DECL E6POS XP526={X 822,Y 549,Z -255,A 0,B -90,C 180,S 6,T 16,E1 0.0,E2 0.0,E3 0.0,E4 0.0,E5 0.0,E6 0.0}
DECL FDAT FP526={TOOL_NO 4,BASE_NO 0,IPO_FRAME #BASE,POINT2[] " "}
DECL LDAT LCPDAT526={VEL 1,ACC 50.000,APO_DIST 500.000,APO_FAC 50.0000,AXIS_VEL 50.000,AXIS_ACC 50.000,ORI_TYP #VAR,CIRC_TYP #BASE,JERK_FAC 50.0000,GEAR_JERK 100.000,EXAX_IGN 0}

DECL E6POS XP527={X 772,Y 549,Z -255,A 0,B -90,C 180,S 6,T 16,E1 0.0,E2 0.0,E3 0.0,E4 0.0,E5 0.0,E6 0.0}
DECL FDAT FP527={TOOL_NO 4,BASE_NO 0,IPO_FRAME #BASE,POINT2[] " "}
DECL LDAT LCPDAT527={VEL 1,ACC 50.000,APO_DIST 500.000,APO_FAC 50.0000,AXIS_VEL 50.000,AXIS_ACC 50.000,ORI_TYP #VAR,CIRC_TYP #BASE,JERK_FAC 50.0000,GEAR_JERK 100.000,EXAX_IGN 0}

DECL E6POS XP528={X 722,Y 549,Z -255,A 0,B -90,C 180,S 6,T 16,E1 0.0,E2 0.0,E3 0.0,E4 0.0,E5 0.0,E6 0.0}
DECL FDAT FP528={TOOL_NO 4,BASE_NO 0,IPO_FRAME #BASE,POINT2[] " "}
DECL LDAT LCPDAT528={VEL 1,ACC 50.000,APO_DIST 500.000,APO_FAC 50.0000,AXIS_VEL 50.000,AXIS_ACC 50.000,ORI_TYP #VAR,CIRC_TYP #BASE,JERK_FAC 50.0000,GEAR_JERK 100.000,EXAX_IGN 0}

DECL E6POS XP529={X 672,Y 549,Z -255,A 0,B -90,C 180,S 6,T 16,E1 0.0,E2 0.0,E3 0.0,E4 0.0,E5 0.0,E6 0.0}
DECL FDAT FP529={TOOL_NO 4,BASE_NO 0,IPO_FRAME #BASE,POINT2[] " "}
DECL LDAT LCPDAT529={VEL 1,ACC 50.000,APO_DIST 500.000,APO_FAC 50.0000,AXIS_VEL 50.000,AXIS_ACC 50.000,ORI_TYP #VAR,CIRC_TYP #BASE,JERK_FAC 50.0000,GEAR_JERK 100.000,EXAX_IGN 0}

DECL E6POS XP530={X 672,Y 549,Z -205,A 0,B -90,C 180,S 6,T 16,E1 0.0,E2 0.0,E3 0.0,E4 0.0,E5 0.0,E6 0.0}
DECL FDAT FP530={TOOL_NO 4,BASE_NO 0,IPO_FRAME #BASE,POINT2[] " "}
DECL LDAT LCPDAT530={VEL 1,ACC 50.000,APO_DIST 500.000,APO_FAC 50.0000,AXIS_VEL 50.000,AXIS_ACC 50.000,ORI_TYP #VAR,CIRC_TYP #BASE,JERK_FAC 50.0000,GEAR_JERK 100.000,EXAX_IGN 0}

DECL E6POS XP531={X 722,Y 549,Z -205,A 0,B -90,C 180,S 6,T 16,E1 0.0,E2 0.0,E3 0.0,E4 0.0,E5 0.0,E6 0.0}
DECL FDAT FP531={TOOL_NO 4,BASE_NO 0,IPO_FRAME #BASE,POINT2[] " "}
DECL LDAT LCPDAT531={VEL 1,ACC 50.000,APO_DIST 500.000,APO_FAC 50.0000,AXIS_VEL 50.000,AXIS_ACC 50.000,ORI_TYP #VAR,CIRC_TYP #BASE,JERK_FAC 50.0000,GEAR_JERK 100.000,EXAX_IGN 0}

DECL E6POS XP532={X 772,Y 549,Z -205,A 0,B -90,C 180,S 6,T 16,E1 0.0,E2 0.0,E3 0.0,E4 0.0,E5 0.0,E6 0.0}
DECL FDAT FP532={TOOL_NO 4,BASE_NO 0,IPO_FRAME #BASE,POINT2[] " "}
DECL LDAT LCPDAT532={VEL 1,ACC 50.000,APO_DIST 500.000,APO_FAC 50.0000,AXIS_VEL 50.000,AXIS_ACC 50.000,ORI_TYP #VAR,CIRC_TYP #BASE,JERK_FAC 50.0000,GEAR_JERK 100.000,EXAX_IGN 0}

DECL E6POS XP533={X 822,Y 549,Z -205,A 0,B -90,C 180,S 6,T 16,E1 0.0,E2 0.0,E3 0.0,E4 0.0,E5 0.0,E6 0.0}
DECL FDAT FP533={TOOL_NO 4,BASE_NO 0,IPO_FRAME #BASE,POINT2[] " "}
DECL LDAT LCPDAT533={VEL 1,ACC 50.000,APO_DIST 500.000,APO_FAC 50.0000,AXIS_VEL 50.000,AXIS_ACC 50.000,ORI_TYP #VAR,CIRC_TYP #BASE,JERK_FAC 50.0000,GEAR_JERK 100.000,EXAX_IGN 0}

DECL E6POS XP534={X 872,Y 549,Z -205,A 0,B -90,C 180,S 6,T 16,E1 0.0,E2 0.0,E3 0.0,E4 0.0,E5 0.0,E6 0.0}
DECL FDAT FP534={TOOL_NO 4,BASE_NO 0,IPO_FRAME #BASE,POINT2[] " "}
DECL LDAT LCPDAT534={VEL 1,ACC 50.000,APO_DIST 500.000,APO_FAC 50.0000,AXIS_VEL 50.000,AXIS_ACC 50.000,ORI_TYP #VAR,CIRC_TYP #BASE,JERK_FAC 50.0000,GEAR_JERK 100.000,EXAX_IGN 0}

DECL E6POS XP535={X 922,Y 549,Z -205,A 0,B -90,C 180,S 6,T 16,E1 0.0,E2 0.0,E3 0.0,E4 0.0,E5 0.0,E6 0.0}
DECL FDAT FP535={TOOL_NO 4,BASE_NO 0,IPO_FRAME #BASE,POINT2[] " "}
DECL LDAT LCPDAT535={VEL 1,ACC 50.000,APO_DIST 500.000,APO_FAC 50.0000,AXIS_VEL 50.000,AXIS_ACC 50.000,ORI_TYP #VAR,CIRC_TYP #BASE,JERK_FAC 50.0000,GEAR_JERK 100.000,EXAX_IGN 0}

DECL E6POS XP536={X 972,Y 549,Z -205,A 0,B -90,C 180,S 6,T 16,E1 0.0,E2 0.0,E3 0.0,E4 0.0,E5 0.0,E6 0.0}
DECL FDAT FP536={TOOL_NO 4,BASE_NO 0,IPO_FRAME #BASE,POINT2[] " "}
DECL LDAT LCPDAT536={VEL 1,ACC 50.000,APO_DIST 500.000,APO_FAC 50.0000,AXIS_VEL 50.000,AXIS_ACC 50.000,ORI_TYP #VAR,CIRC_TYP #BASE,JERK_FAC 50.0000,GEAR_JERK 100.000,EXAX_IGN 0}

DECL E6POS XP537={X 1022,Y 549,Z -205,A 0,B -90,C 180,S 6,T 16,E1 0.0,E2 0.0,E3 0.0,E4 0.0,E5 0.0,E6 0.0}
DECL FDAT FP537={TOOL_NO 4,BASE_NO 0,IPO_FRAME #BASE,POINT2[] " "}
DECL LDAT LCPDAT537={VEL 1,ACC 50.000,APO_DIST 500.000,APO_FAC 50.0000,AXIS_VEL 50.000,AXIS_ACC 50.000,ORI_TYP #VAR,CIRC_TYP #BASE,JERK_FAC 50.0000,GEAR_JERK 100.000,EXAX_IGN 0}

DECL E6POS XP538={X 1072,Y 549,Z -205,A 0,B -90,C 180,S 6,T 16,E1 0.0,E2 0.0,E3 0.0,E4 0.0,E5 0.0,E6 0.0}
DECL FDAT FP538={TOOL_NO 4,BASE_NO 0,IPO_FRAME #BASE,POINT2[] " "}
DECL LDAT LCPDAT538={VEL 1,ACC 50.000,APO_DIST 500.000,APO_FAC 50.0000,AXIS_VEL 50.000,AXIS_ACC 50.000,ORI_TYP #VAR,CIRC_TYP #BASE,JERK_FAC 50.0000,GEAR_JERK 100.000,EXAX_IGN 0}

DECL E6POS XP539={X 1122,Y 549,Z -205,A 0,B -90,C 180,S 6,T 16,E1 0.0,E2 0.0,E3 0.0,E4 0.0,E5 0.0,E6 0.0}
DECL FDAT FP539={TOOL_NO 4,BASE_NO 0,IPO_FRAME #BASE,POINT2[] " "}
DECL LDAT LCPDAT539={VEL 1,ACC 50.000,APO_DIST 500.000,APO_FAC 50.0000,AXIS_VEL 50.000,AXIS_ACC 50.000,ORI_TYP #VAR,CIRC_TYP #BASE,JERK_FAC 50.0000,GEAR_JERK 100.000,EXAX_IGN 0}

DECL E6POS XP540={X 1172,Y 549,Z -205,A 0,B -90,C 180,S 6,T 16,E1 0.0,E2 0.0,E3 0.0,E4 0.0,E5 0.0,E6 0.0}
DECL FDAT FP540={TOOL_NO 4,BASE_NO 0,IPO_FRAME #BASE,POINT2[] " "}
DECL LDAT LCPDAT540={VEL 1,ACC 50.000,APO_DIST 500.000,APO_FAC 50.0000,AXIS_VEL 50.000,AXIS_ACC 50.000,ORI_TYP #VAR,CIRC_TYP #BASE,JERK_FAC 50.0000,GEAR_JERK 100.000,EXAX_IGN 0}

DECL E6POS XP541={X 1222,Y 549,Z -205,A 0,B -90,C 180,S 6,T 16,E1 0.0,E2 0.0,E3 0.0,E4 0.0,E5 0.0,E6 0.0}
DECL FDAT FP541={TOOL_NO 4,BASE_NO 0,IPO_FRAME #BASE,POINT2[] " "}
DECL LDAT LCPDAT541={VEL 1,ACC 50.000,APO_DIST 500.000,APO_FAC 50.0000,AXIS_VEL 50.000,AXIS_ACC 50.000,ORI_TYP #VAR,CIRC_TYP #BASE,JERK_FAC 50.0000,GEAR_JERK 100.000,EXAX_IGN 0}

DECL E6POS XP542={X 1272,Y 549,Z -205,A 0,B -90,C 180,S 6,T 16,E1 0.0,E2 0.0,E3 0.0,E4 0.0,E5 0.0,E6 0.0}
DECL FDAT FP542={TOOL_NO 4,BASE_NO 0,IPO_FRAME #BASE,POINT2[] " "}
DECL LDAT LCPDAT542={VEL 1,ACC 50.000,APO_DIST 500.000,APO_FAC 50.0000,AXIS_VEL 50.000,AXIS_ACC 50.000,ORI_TYP #VAR,CIRC_TYP #BASE,JERK_FAC 50.0000,GEAR_JERK 100.000,EXAX_IGN 0}

DECL E6POS XP543={X 1272,Y 549,Z -155,A 0,B -90,C 180,S 6,T 16,E1 0.0,E2 0.0,E3 0.0,E4 0.0,E5 0.0,E6 0.0}
DECL FDAT FP543={TOOL_NO 4,BASE_NO 0,IPO_FRAME #BASE,POINT2[] " "}
DECL LDAT LCPDAT543={VEL 1,ACC 50.000,APO_DIST 500.000,APO_FAC 50.0000,AXIS_VEL 50.000,AXIS_ACC 50.000,ORI_TYP #VAR,CIRC_TYP #BASE,JERK_FAC 50.0000,GEAR_JERK 100.000,EXAX_IGN 0}

DECL E6POS XP544={X 1222,Y 549,Z -155,A 0,B -90,C 180,S 6,T 16,E1 0.0,E2 0.0,E3 0.0,E4 0.0,E5 0.0,E6 0.0}
DECL FDAT FP544={TOOL_NO 4,BASE_NO 0,IPO_FRAME #BASE,POINT2[] " "}
DECL LDAT LCPDAT544={VEL 1,ACC 50.000,APO_DIST 500.000,APO_FAC 50.0000,AXIS_VEL 50.000,AXIS_ACC 50.000,ORI_TYP #VAR,CIRC_TYP #BASE,JERK_FAC 50.0000,GEAR_JERK 100.000,EXAX_IGN 0}

DECL E6POS XP545={X 1172,Y 549,Z -155,A 0,B -90,C 180,S 6,T 16,E1 0.0,E2 0.0,E3 0.0,E4 0.0,E5 0.0,E6 0.0}
DECL FDAT FP545={TOOL_NO 4,BASE_NO 0,IPO_FRAME #BASE,POINT2[] " "}
DECL LDAT LCPDAT545={VEL 1,ACC 50.000,APO_DIST 500.000,APO_FAC 50.0000,AXIS_VEL 50.000,AXIS_ACC 50.000,ORI_TYP #VAR,CIRC_TYP #BASE,JERK_FAC 50.0000,GEAR_JERK 100.000,EXAX_IGN 0}

DECL E6POS XP546={X 1122,Y 549,Z -155,A 0,B -90,C 180,S 6,T 16,E1 0.0,E2 0.0,E3 0.0,E4 0.0,E5 0.0,E6 0.0}
DECL FDAT FP546={TOOL_NO 4,BASE_NO 0,IPO_FRAME #BASE,POINT2[] " "}
DECL LDAT LCPDAT546={VEL 1,ACC 50.000,APO_DIST 500.000,APO_FAC 50.0000,AXIS_VEL 50.000,AXIS_ACC 50.000,ORI_TYP #VAR,CIRC_TYP #BASE,JERK_FAC 50.0000,GEAR_JERK 100.000,EXAX_IGN 0}

DECL E6POS XP547={X 1072,Y 549,Z -155,A 0,B -90,C 180,S 6,T 16,E1 0.0,E2 0.0,E3 0.0,E4 0.0,E5 0.0,E6 0.0}
DECL FDAT FP547={TOOL_NO 4,BASE_NO 0,IPO_FRAME #BASE,POINT2[] " "}
DECL LDAT LCPDAT547={VEL 1,ACC 50.000,APO_DIST 500.000,APO_FAC 50.0000,AXIS_VEL 50.000,AXIS_ACC 50.000,ORI_TYP #VAR,CIRC_TYP #BASE,JERK_FAC 50.0000,GEAR_JERK 100.000,EXAX_IGN 0}

DECL E6POS XP548={X 1022,Y 549,Z -155,A 0,B -90,C 180,S 6,T 16,E1 0.0,E2 0.0,E3 0.0,E4 0.0,E5 0.0,E6 0.0}
DECL FDAT FP548={TOOL_NO 4,BASE_NO 0,IPO_FRAME #BASE,POINT2[] " "}
DECL LDAT LCPDAT548={VEL 1,ACC 50.000,APO_DIST 500.000,APO_FAC 50.0000,AXIS_VEL 50.000,AXIS_ACC 50.000,ORI_TYP #VAR,CIRC_TYP #BASE,JERK_FAC 50.0000,GEAR_JERK 100.000,EXAX_IGN 0}

DECL E6POS XP549={X 972,Y 549,Z -155,A 0,B -90,C 180,S 6,T 16,E1 0.0,E2 0.0,E3 0.0,E4 0.0,E5 0.0,E6 0.0}
DECL FDAT FP549={TOOL_NO 4,BASE_NO 0,IPO_FRAME #BASE,POINT2[] " "}
DECL LDAT LCPDAT549={VEL 1,ACC 50.000,APO_DIST 500.000,APO_FAC 50.0000,AXIS_VEL 50.000,AXIS_ACC 50.000,ORI_TYP #VAR,CIRC_TYP #BASE,JERK_FAC 50.0000,GEAR_JERK 100.000,EXAX_IGN 0}

DECL E6POS XP550={X 922,Y 549,Z -155,A 0,B -90,C 180,S 6,T 16,E1 0.0,E2 0.0,E3 0.0,E4 0.0,E5 0.0,E6 0.0}
DECL FDAT FP550={TOOL_NO 4,BASE_NO 0,IPO_FRAME #BASE,POINT2[] " "}
DECL LDAT LCPDAT550={VEL 1,ACC 50.000,APO_DIST 500.000,APO_FAC 50.0000,AXIS_VEL 50.000,AXIS_ACC 50.000,ORI_TYP #VAR,CIRC_TYP #BASE,JERK_FAC 50.0000,GEAR_JERK 100.000,EXAX_IGN 0}

DECL E6POS XP551={X 872,Y 549,Z -155,A 0,B -90,C 180,S 6,T 16,E1 0.0,E2 0.0,E3 0.0,E4 0.0,E5 0.0,E6 0.0}
DECL FDAT FP551={TOOL_NO 4,BASE_NO 0,IPO_FRAME #BASE,POINT2[] " "}
DECL LDAT LCPDAT551={VEL 1,ACC 50.000,APO_DIST 500.000,APO_FAC 50.0000,AXIS_VEL 50.000,AXIS_ACC 50.000,ORI_TYP #VAR,CIRC_TYP #BASE,JERK_FAC 50.0000,GEAR_JERK 100.000,EXAX_IGN 0}

DECL E6POS XP552={X 822,Y 549,Z -155,A 0,B -90,C 180,S 6,T 16,E1 0.0,E2 0.0,E3 0.0,E4 0.0,E5 0.0,E6 0.0}
DECL FDAT FP552={TOOL_NO 4,BASE_NO 0,IPO_FRAME #BASE,POINT2[] " "}
DECL LDAT LCPDAT552={VEL 1,ACC 50.000,APO_DIST 500.000,APO_FAC 50.0000,AXIS_VEL 50.000,AXIS_ACC 50.000,ORI_TYP #VAR,CIRC_TYP #BASE,JERK_FAC 50.0000,GEAR_JERK 100.000,EXAX_IGN 0}

DECL E6POS XP553={X 772,Y 549,Z -155,A 0,B -90,C 180,S 6,T 16,E1 0.0,E2 0.0,E3 0.0,E4 0.0,E5 0.0,E6 0.0}
DECL FDAT FP553={TOOL_NO 4,BASE_NO 0,IPO_FRAME #BASE,POINT2[] " "}
DECL LDAT LCPDAT553={VEL 1,ACC 50.000,APO_DIST 500.000,APO_FAC 50.0000,AXIS_VEL 50.000,AXIS_ACC 50.000,ORI_TYP #VAR,CIRC_TYP #BASE,JERK_FAC 50.0000,GEAR_JERK 100.000,EXAX_IGN 0}

DECL E6POS XP554={X 722,Y 549,Z -155,A 0,B -90,C 180,S 6,T 16,E1 0.0,E2 0.0,E3 0.0,E4 0.0,E5 0.0,E6 0.0}
DECL FDAT FP554={TOOL_NO 4,BASE_NO 0,IPO_FRAME #BASE,POINT2[] " "}
DECL LDAT LCPDAT554={VEL 1,ACC 50.000,APO_DIST 500.000,APO_FAC 50.0000,AXIS_VEL 50.000,AXIS_ACC 50.000,ORI_TYP #VAR,CIRC_TYP #BASE,JERK_FAC 50.0000,GEAR_JERK 100.000,EXAX_IGN 0}

DECL E6POS XP555={X 672,Y 549,Z -155,A 0,B -90,C 180,S 6,T 16,E1 0.0,E2 0.0,E3 0.0,E4 0.0,E5 0.0,E6 0.0}
DECL FDAT FP555={TOOL_NO 4,BASE_NO 0,IPO_FRAME #BASE,POINT2[] " "}
DECL LDAT LCPDAT555={VEL 1,ACC 50.000,APO_DIST 500.000,APO_FAC 50.0000,AXIS_VEL 50.000,AXIS_ACC 50.000,ORI_TYP #VAR,CIRC_TYP #BASE,JERK_FAC 50.0000,GEAR_JERK 100.000,EXAX_IGN 0}

DECL E6POS XP556={X 672,Y 549,Z -105,A 0,B -90,C 180,S 6,T 16,E1 0.0,E2 0.0,E3 0.0,E4 0.0,E5 0.0,E6 0.0}
DECL FDAT FP556={TOOL_NO 4,BASE_NO 0,IPO_FRAME #BASE,POINT2[] " "}
DECL LDAT LCPDAT556={VEL 1,ACC 50.000,APO_DIST 500.000,APO_FAC 50.0000,AXIS_VEL 50.000,AXIS_ACC 50.000,ORI_TYP #VAR,CIRC_TYP #BASE,JERK_FAC 50.0000,GEAR_JERK 100.000,EXAX_IGN 0}

DECL E6POS XP557={X 722,Y 549,Z -105,A 0,B -90,C 180,S 6,T 16,E1 0.0,E2 0.0,E3 0.0,E4 0.0,E5 0.0,E6 0.0}
DECL FDAT FP557={TOOL_NO 4,BASE_NO 0,IPO_FRAME #BASE,POINT2[] " "}
DECL LDAT LCPDAT557={VEL 1,ACC 50.000,APO_DIST 500.000,APO_FAC 50.0000,AXIS_VEL 50.000,AXIS_ACC 50.000,ORI_TYP #VAR,CIRC_TYP #BASE,JERK_FAC 50.0000,GEAR_JERK 100.000,EXAX_IGN 0}

DECL E6POS XP558={X 772,Y 549,Z -105,A 0,B -90,C 180,S 6,T 16,E1 0.0,E2 0.0,E3 0.0,E4 0.0,E5 0.0,E6 0.0}
DECL FDAT FP558={TOOL_NO 4,BASE_NO 0,IPO_FRAME #BASE,POINT2[] " "}
DECL LDAT LCPDAT558={VEL 1,ACC 50.000,APO_DIST 500.000,APO_FAC 50.0000,AXIS_VEL 50.000,AXIS_ACC 50.000,ORI_TYP #VAR,CIRC_TYP #BASE,JERK_FAC 50.0000,GEAR_JERK 100.000,EXAX_IGN 0}

DECL E6POS XP559={X 822,Y 549,Z -105,A 0,B -90,C 180,S 6,T 16,E1 0.0,E2 0.0,E3 0.0,E4 0.0,E5 0.0,E6 0.0}
DECL FDAT FP559={TOOL_NO 4,BASE_NO 0,IPO_FRAME #BASE,POINT2[] " "}
DECL LDAT LCPDAT559={VEL 1,ACC 50.000,APO_DIST 500.000,APO_FAC 50.0000,AXIS_VEL 50.000,AXIS_ACC 50.000,ORI_TYP #VAR,CIRC_TYP #BASE,JERK_FAC 50.0000,GEAR_JERK 100.000,EXAX_IGN 0}

DECL E6POS XP560={X 872,Y 549,Z -105,A 0,B -90,C 180,S 6,T 16,E1 0.0,E2 0.0,E3 0.0,E4 0.0,E5 0.0,E6 0.0}
DECL FDAT FP560={TOOL_NO 4,BASE_NO 0,IPO_FRAME #BASE,POINT2[] " "}
DECL LDAT LCPDAT560={VEL 1,ACC 50.000,APO_DIST 500.000,APO_FAC 50.0000,AXIS_VEL 50.000,AXIS_ACC 50.000,ORI_TYP #VAR,CIRC_TYP #BASE,JERK_FAC 50.0000,GEAR_JERK 100.000,EXAX_IGN 0}

DECL E6POS XP561={X 922,Y 549,Z -105,A 0,B -90,C 180,S 6,T 16,E1 0.0,E2 0.0,E3 0.0,E4 0.0,E5 0.0,E6 0.0}
DECL FDAT FP561={TOOL_NO 4,BASE_NO 0,IPO_FRAME #BASE,POINT2[] " "}
DECL LDAT LCPDAT561={VEL 1,ACC 50.000,APO_DIST 500.000,APO_FAC 50.0000,AXIS_VEL 50.000,AXIS_ACC 50.000,ORI_TYP #VAR,CIRC_TYP #BASE,JERK_FAC 50.0000,GEAR_JERK 100.000,EXAX_IGN 0}

DECL E6POS XP562={X 972,Y 549,Z -105,A 0,B -90,C 180,S 6,T 16,E1 0.0,E2 0.0,E3 0.0,E4 0.0,E5 0.0,E6 0.0}
DECL FDAT FP562={TOOL_NO 4,BASE_NO 0,IPO_FRAME #BASE,POINT2[] " "}
DECL LDAT LCPDAT562={VEL 1,ACC 50.000,APO_DIST 500.000,APO_FAC 50.0000,AXIS_VEL 50.000,AXIS_ACC 50.000,ORI_TYP #VAR,CIRC_TYP #BASE,JERK_FAC 50.0000,GEAR_JERK 100.000,EXAX_IGN 0}

DECL E6POS XP563={X 1022,Y 549,Z -105,A 0,B -90,C 180,S 6,T 16,E1 0.0,E2 0.0,E3 0.0,E4 0.0,E5 0.0,E6 0.0}
DECL FDAT FP563={TOOL_NO 4,BASE_NO 0,IPO_FRAME #BASE,POINT2[] " "}
DECL LDAT LCPDAT563={VEL 1,ACC 50.000,APO_DIST 500.000,APO_FAC 50.0000,AXIS_VEL 50.000,AXIS_ACC 50.000,ORI_TYP #VAR,CIRC_TYP #BASE,JERK_FAC 50.0000,GEAR_JERK 100.000,EXAX_IGN 0}

DECL E6POS XP564={X 1072,Y 549,Z -105,A 0,B -90,C 180,S 6,T 16,E1 0.0,E2 0.0,E3 0.0,E4 0.0,E5 0.0,E6 0.0}
DECL FDAT FP564={TOOL_NO 4,BASE_NO 0,IPO_FRAME #BASE,POINT2[] " "}
DECL LDAT LCPDAT564={VEL 1,ACC 50.000,APO_DIST 500.000,APO_FAC 50.0000,AXIS_VEL 50.000,AXIS_ACC 50.000,ORI_TYP #VAR,CIRC_TYP #BASE,JERK_FAC 50.0000,GEAR_JERK 100.000,EXAX_IGN 0}

DECL E6POS XP565={X 1122,Y 549,Z -105,A 0,B -90,C 180,S 6,T 16,E1 0.0,E2 0.0,E3 0.0,E4 0.0,E5 0.0,E6 0.0}
DECL FDAT FP565={TOOL_NO 4,BASE_NO 0,IPO_FRAME #BASE,POINT2[] " "}
DECL LDAT LCPDAT565={VEL 1,ACC 50.000,APO_DIST 500.000,APO_FAC 50.0000,AXIS_VEL 50.000,AXIS_ACC 50.000,ORI_TYP #VAR,CIRC_TYP #BASE,JERK_FAC 50.0000,GEAR_JERK 100.000,EXAX_IGN 0}

DECL E6POS XP566={X 1172,Y 549,Z -105,A 0,B -90,C 180,S 6,T 16,E1 0.0,E2 0.0,E3 0.0,E4 0.0,E5 0.0,E6 0.0}
DECL FDAT FP566={TOOL_NO 4,BASE_NO 0,IPO_FRAME #BASE,POINT2[] " "}
DECL LDAT LCPDAT566={VEL 1,ACC 50.000,APO_DIST 500.000,APO_FAC 50.0000,AXIS_VEL 50.000,AXIS_ACC 50.000,ORI_TYP #VAR,CIRC_TYP #BASE,JERK_FAC 50.0000,GEAR_JERK 100.000,EXAX_IGN 0}

DECL E6POS XP567={X 1222,Y 549,Z -105,A 0,B -90,C 180,S 6,T 16,E1 0.0,E2 0.0,E3 0.0,E4 0.0,E5 0.0,E6 0.0}
DECL FDAT FP567={TOOL_NO 4,BASE_NO 0,IPO_FRAME #BASE,POINT2[] " "}
DECL LDAT LCPDAT567={VEL 1,ACC 50.000,APO_DIST 500.000,APO_FAC 50.0000,AXIS_VEL 50.000,AXIS_ACC 50.000,ORI_TYP #VAR,CIRC_TYP #BASE,JERK_FAC 50.0000,GEAR_JERK 100.000,EXAX_IGN 0}

DECL E6POS XP568={X 1272,Y 549,Z -105,A 0,B -90,C 180,S 6,T 16,E1 0.0,E2 0.0,E3 0.0,E4 0.0,E5 0.0,E6 0.0}
DECL FDAT FP568={TOOL_NO 4,BASE_NO 0,IPO_FRAME #BASE,POINT2[] " "}
DECL LDAT LCPDAT568={VEL 1,ACC 50.000,APO_DIST 500.000,APO_FAC 50.0000,AXIS_VEL 50.000,AXIS_ACC 50.000,ORI_TYP #VAR,CIRC_TYP #BASE,JERK_FAC 50.0000,GEAR_JERK 100.000,EXAX_IGN 0}

DECL E6POS XP569={X 1272,Y 549,Z -55,A 0,B -90,C 180,S 6,T 16,E1 0.0,E2 0.0,E3 0.0,E4 0.0,E5 0.0,E6 0.0}
DECL FDAT FP569={TOOL_NO 4,BASE_NO 0,IPO_FRAME #BASE,POINT2[] " "}
DECL LDAT LCPDAT569={VEL 1,ACC 50.000,APO_DIST 500.000,APO_FAC 50.0000,AXIS_VEL 50.000,AXIS_ACC 50.000,ORI_TYP #VAR,CIRC_TYP #BASE,JERK_FAC 50.0000,GEAR_JERK 100.000,EXAX_IGN 0}

DECL E6POS XP570={X 1222,Y 549,Z -55,A 0,B -90,C 180,S 6,T 16,E1 0.0,E2 0.0,E3 0.0,E4 0.0,E5 0.0,E6 0.0}
DECL FDAT FP570={TOOL_NO 4,BASE_NO 0,IPO_FRAME #BASE,POINT2[] " "}
DECL LDAT LCPDAT570={VEL 1,ACC 50.000,APO_DIST 500.000,APO_FAC 50.0000,AXIS_VEL 50.000,AXIS_ACC 50.000,ORI_TYP #VAR,CIRC_TYP #BASE,JERK_FAC 50.0000,GEAR_JERK 100.000,EXAX_IGN 0}

DECL E6POS XP571={X 1172,Y 549,Z -55,A 0,B -90,C 180,S 6,T 16,E1 0.0,E2 0.0,E3 0.0,E4 0.0,E5 0.0,E6 0.0}
DECL FDAT FP571={TOOL_NO 4,BASE_NO 0,IPO_FRAME #BASE,POINT2[] " "}
DECL LDAT LCPDAT571={VEL 1,ACC 50.000,APO_DIST 500.000,APO_FAC 50.0000,AXIS_VEL 50.000,AXIS_ACC 50.000,ORI_TYP #VAR,CIRC_TYP #BASE,JERK_FAC 50.0000,GEAR_JERK 100.000,EXAX_IGN 0}

DECL E6POS XP572={X 1122,Y 549,Z -55,A 0,B -90,C 180,S 6,T 16,E1 0.0,E2 0.0,E3 0.0,E4 0.0,E5 0.0,E6 0.0}
DECL FDAT FP572={TOOL_NO 4,BASE_NO 0,IPO_FRAME #BASE,POINT2[] " "}
DECL LDAT LCPDAT572={VEL 1,ACC 50.000,APO_DIST 500.000,APO_FAC 50.0000,AXIS_VEL 50.000,AXIS_ACC 50.000,ORI_TYP #VAR,CIRC_TYP #BASE,JERK_FAC 50.0000,GEAR_JERK 100.000,EXAX_IGN 0}

DECL E6POS XP573={X 1072,Y 549,Z -55,A 0,B -90,C 180,S 6,T 16,E1 0.0,E2 0.0,E3 0.0,E4 0.0,E5 0.0,E6 0.0}
DECL FDAT FP573={TOOL_NO 4,BASE_NO 0,IPO_FRAME #BASE,POINT2[] " "}
DECL LDAT LCPDAT573={VEL 1,ACC 50.000,APO_DIST 500.000,APO_FAC 50.0000,AXIS_VEL 50.000,AXIS_ACC 50.000,ORI_TYP #VAR,CIRC_TYP #BASE,JERK_FAC 50.0000,GEAR_JERK 100.000,EXAX_IGN 0}

DECL E6POS XP574={X 1022,Y 549,Z -55,A 0,B -90,C 180,S 6,T 16,E1 0.0,E2 0.0,E3 0.0,E4 0.0,E5 0.0,E6 0.0}
DECL FDAT FP574={TOOL_NO 4,BASE_NO 0,IPO_FRAME #BASE,POINT2[] " "}
DECL LDAT LCPDAT574={VEL 1,ACC 50.000,APO_DIST 500.000,APO_FAC 50.0000,AXIS_VEL 50.000,AXIS_ACC 50.000,ORI_TYP #VAR,CIRC_TYP #BASE,JERK_FAC 50.0000,GEAR_JERK 100.000,EXAX_IGN 0}

DECL E6POS XP575={X 972,Y 549,Z -55,A 0,B -90,C 180,S 6,T 16,E1 0.0,E2 0.0,E3 0.0,E4 0.0,E5 0.0,E6 0.0}
DECL FDAT FP575={TOOL_NO 4,BASE_NO 0,IPO_FRAME #BASE,POINT2[] " "}
DECL LDAT LCPDAT575={VEL 1,ACC 50.000,APO_DIST 500.000,APO_FAC 50.0000,AXIS_VEL 50.000,AXIS_ACC 50.000,ORI_TYP #VAR,CIRC_TYP #BASE,JERK_FAC 50.0000,GEAR_JERK 100.000,EXAX_IGN 0}

DECL E6POS XP576={X 922,Y 549,Z -55,A 0,B -90,C 180,S 6,T 16,E1 0.0,E2 0.0,E3 0.0,E4 0.0,E5 0.0,E6 0.0}
DECL FDAT FP576={TOOL_NO 4,BASE_NO 0,IPO_FRAME #BASE,POINT2[] " "}
DECL LDAT LCPDAT576={VEL 1,ACC 50.000,APO_DIST 500.000,APO_FAC 50.0000,AXIS_VEL 50.000,AXIS_ACC 50.000,ORI_TYP #VAR,CIRC_TYP #BASE,JERK_FAC 50.0000,GEAR_JERK 100.000,EXAX_IGN 0}

DECL E6POS XP577={X 872,Y 549,Z -55,A 0,B -90,C 180,S 6,T 16,E1 0.0,E2 0.0,E3 0.0,E4 0.0,E5 0.0,E6 0.0}
DECL FDAT FP577={TOOL_NO 4,BASE_NO 0,IPO_FRAME #BASE,POINT2[] " "}
DECL LDAT LCPDAT577={VEL 1,ACC 50.000,APO_DIST 500.000,APO_FAC 50.0000,AXIS_VEL 50.000,AXIS_ACC 50.000,ORI_TYP #VAR,CIRC_TYP #BASE,JERK_FAC 50.0000,GEAR_JERK 100.000,EXAX_IGN 0}

DECL E6POS XP578={X 822,Y 549,Z -55,A 0,B -90,C 180,S 6,T 16,E1 0.0,E2 0.0,E3 0.0,E4 0.0,E5 0.0,E6 0.0}
DECL FDAT FP578={TOOL_NO 4,BASE_NO 0,IPO_FRAME #BASE,POINT2[] " "}
DECL LDAT LCPDAT578={VEL 1,ACC 50.000,APO_DIST 500.000,APO_FAC 50.0000,AXIS_VEL 50.000,AXIS_ACC 50.000,ORI_TYP #VAR,CIRC_TYP #BASE,JERK_FAC 50.0000,GEAR_JERK 100.000,EXAX_IGN 0}

DECL E6POS XP579={X 772,Y 549,Z -55,A 0,B -90,C 180,S 6,T 16,E1 0.0,E2 0.0,E3 0.0,E4 0.0,E5 0.0,E6 0.0}
DECL FDAT FP579={TOOL_NO 4,BASE_NO 0,IPO_FRAME #BASE,POINT2[] " "}
DECL LDAT LCPDAT579={VEL 1,ACC 50.000,APO_DIST 500.000,APO_FAC 50.0000,AXIS_VEL 50.000,AXIS_ACC 50.000,ORI_TYP #VAR,CIRC_TYP #BASE,JERK_FAC 50.0000,GEAR_JERK 100.000,EXAX_IGN 0}

DECL E6POS XP580={X 722,Y 549,Z -55,A 0,B -90,C 180,S 6,T 16,E1 0.0,E2 0.0,E3 0.0,E4 0.0,E5 0.0,E6 0.0}
DECL FDAT FP580={TOOL_NO 4,BASE_NO 0,IPO_FRAME #BASE,POINT2[] " "}
DECL LDAT LCPDAT580={VEL 1,ACC 50.000,APO_DIST 500.000,APO_FAC 50.0000,AXIS_VEL 50.000,AXIS_ACC 50.000,ORI_TYP #VAR,CIRC_TYP #BASE,JERK_FAC 50.0000,GEAR_JERK 100.000,EXAX_IGN 0}

DECL E6POS XP581={X 672,Y 549,Z -55,A 0,B -90,C 180,S 6,T 16,E1 0.0,E2 0.0,E3 0.0,E4 0.0,E5 0.0,E6 0.0}
DECL FDAT FP581={TOOL_NO 4,BASE_NO 0,IPO_FRAME #BASE,POINT2[] " "}
DECL LDAT LCPDAT581={VEL 1,ACC 50.000,APO_DIST 500.000,APO_FAC 50.0000,AXIS_VEL 50.000,AXIS_ACC 50.000,ORI_TYP #VAR,CIRC_TYP #BASE,JERK_FAC 50.0000,GEAR_JERK 100.000,EXAX_IGN 0}

DECL E6POS XP582={X 672,Y 549,Z -5,A 0,B -90,C 180,S 6,T 16,E1 0.0,E2 0.0,E3 0.0,E4 0.0,E5 0.0,E6 0.0}
DECL FDAT FP582={TOOL_NO 4,BASE_NO 0,IPO_FRAME #BASE,POINT2[] " "}
DECL LDAT LCPDAT582={VEL 1,ACC 50.000,APO_DIST 500.000,APO_FAC 50.0000,AXIS_VEL 50.000,AXIS_ACC 50.000,ORI_TYP #VAR,CIRC_TYP #BASE,JERK_FAC 50.0000,GEAR_JERK 100.000,EXAX_IGN 0}

DECL E6POS XP583={X 722,Y 549,Z -5,A 0,B -90,C 180,S 6,T 16,E1 0.0,E2 0.0,E3 0.0,E4 0.0,E5 0.0,E6 0.0}
DECL FDAT FP583={TOOL_NO 4,BASE_NO 0,IPO_FRAME #BASE,POINT2[] " "}
DECL LDAT LCPDAT583={VEL 1,ACC 50.000,APO_DIST 500.000,APO_FAC 50.0000,AXIS_VEL 50.000,AXIS_ACC 50.000,ORI_TYP #VAR,CIRC_TYP #BASE,JERK_FAC 50.0000,GEAR_JERK 100.000,EXAX_IGN 0}

DECL E6POS XP584={X 772,Y 549,Z -5,A 0,B -90,C 180,S 6,T 16,E1 0.0,E2 0.0,E3 0.0,E4 0.0,E5 0.0,E6 0.0}
DECL FDAT FP584={TOOL_NO 4,BASE_NO 0,IPO_FRAME #BASE,POINT2[] " "}
DECL LDAT LCPDAT584={VEL 1,ACC 50.000,APO_DIST 500.000,APO_FAC 50.0000,AXIS_VEL 50.000,AXIS_ACC 50.000,ORI_TYP #VAR,CIRC_TYP #BASE,JERK_FAC 50.0000,GEAR_JERK 100.000,EXAX_IGN 0}

DECL E6POS XP585={X 822,Y 549,Z -5,A 0,B -90,C 180,S 6,T 16,E1 0.0,E2 0.0,E3 0.0,E4 0.0,E5 0.0,E6 0.0}
DECL FDAT FP585={TOOL_NO 4,BASE_NO 0,IPO_FRAME #BASE,POINT2[] " "}
DECL LDAT LCPDAT585={VEL 1,ACC 50.000,APO_DIST 500.000,APO_FAC 50.0000,AXIS_VEL 50.000,AXIS_ACC 50.000,ORI_TYP #VAR,CIRC_TYP #BASE,JERK_FAC 50.0000,GEAR_JERK 100.000,EXAX_IGN 0}

DECL E6POS XP586={X 872,Y 549,Z -5,A 0,B -90,C 180,S 6,T 16,E1 0.0,E2 0.0,E3 0.0,E4 0.0,E5 0.0,E6 0.0}
DECL FDAT FP586={TOOL_NO 4,BASE_NO 0,IPO_FRAME #BASE,POINT2[] " "}
DECL LDAT LCPDAT586={VEL 1,ACC 50.000,APO_DIST 500.000,APO_FAC 50.0000,AXIS_VEL 50.000,AXIS_ACC 50.000,ORI_TYP #VAR,CIRC_TYP #BASE,JERK_FAC 50.0000,GEAR_JERK 100.000,EXAX_IGN 0}

DECL E6POS XP587={X 922,Y 549,Z -5,A 0,B -90,C 180,S 6,T 16,E1 0.0,E2 0.0,E3 0.0,E4 0.0,E5 0.0,E6 0.0}
DECL FDAT FP587={TOOL_NO 4,BASE_NO 0,IPO_FRAME #BASE,POINT2[] " "}
DECL LDAT LCPDAT587={VEL 1,ACC 50.000,APO_DIST 500.000,APO_FAC 50.0000,AXIS_VEL 50.000,AXIS_ACC 50.000,ORI_TYP #VAR,CIRC_TYP #BASE,JERK_FAC 50.0000,GEAR_JERK 100.000,EXAX_IGN 0}

DECL E6POS XP588={X 972,Y 549,Z -5,A 0,B -90,C 180,S 6,T 16,E1 0.0,E2 0.0,E3 0.0,E4 0.0,E5 0.0,E6 0.0}
DECL FDAT FP588={TOOL_NO 4,BASE_NO 0,IPO_FRAME #BASE,POINT2[] " "}
DECL LDAT LCPDAT588={VEL 1,ACC 50.000,APO_DIST 500.000,APO_FAC 50.0000,AXIS_VEL 50.000,AXIS_ACC 50.000,ORI_TYP #VAR,CIRC_TYP #BASE,JERK_FAC 50.0000,GEAR_JERK 100.000,EXAX_IGN 0}

DECL E6POS XP589={X 1022,Y 549,Z -5,A 0,B -90,C 180,S 6,T 16,E1 0.0,E2 0.0,E3 0.0,E4 0.0,E5 0.0,E6 0.0}
DECL FDAT FP589={TOOL_NO 4,BASE_NO 0,IPO_FRAME #BASE,POINT2[] " "}
DECL LDAT LCPDAT589={VEL 1,ACC 50.000,APO_DIST 500.000,APO_FAC 50.0000,AXIS_VEL 50.000,AXIS_ACC 50.000,ORI_TYP #VAR,CIRC_TYP #BASE,JERK_FAC 50.0000,GEAR_JERK 100.000,EXAX_IGN 0}

DECL E6POS XP590={X 1072,Y 549,Z -5,A 0,B -90,C 180,S 6,T 16,E1 0.0,E2 0.0,E3 0.0,E4 0.0,E5 0.0,E6 0.0}
DECL FDAT FP590={TOOL_NO 4,BASE_NO 0,IPO_FRAME #BASE,POINT2[] " "}
DECL LDAT LCPDAT590={VEL 1,ACC 50.000,APO_DIST 500.000,APO_FAC 50.0000,AXIS_VEL 50.000,AXIS_ACC 50.000,ORI_TYP #VAR,CIRC_TYP #BASE,JERK_FAC 50.0000,GEAR_JERK 100.000,EXAX_IGN 0}

DECL E6POS XP591={X 1122,Y 549,Z -5,A 0,B -90,C 180,S 6,T 16,E1 0.0,E2 0.0,E3 0.0,E4 0.0,E5 0.0,E6 0.0}
DECL FDAT FP591={TOOL_NO 4,BASE_NO 0,IPO_FRAME #BASE,POINT2[] " "}
DECL LDAT LCPDAT591={VEL 1,ACC 50.000,APO_DIST 500.000,APO_FAC 50.0000,AXIS_VEL 50.000,AXIS_ACC 50.000,ORI_TYP #VAR,CIRC_TYP #BASE,JERK_FAC 50.0000,GEAR_JERK 100.000,EXAX_IGN 0}

DECL E6POS XP592={X 1172,Y 549,Z -5,A 0,B -90,C 180,S 6,T 16,E1 0.0,E2 0.0,E3 0.0,E4 0.0,E5 0.0,E6 0.0}
DECL FDAT FP592={TOOL_NO 4,BASE_NO 0,IPO_FRAME #BASE,POINT2[] " "}
DECL LDAT LCPDAT592={VEL 1,ACC 50.000,APO_DIST 500.000,APO_FAC 50.0000,AXIS_VEL 50.000,AXIS_ACC 50.000,ORI_TYP #VAR,CIRC_TYP #BASE,JERK_FAC 50.0000,GEAR_JERK 100.000,EXAX_IGN 0}

DECL E6POS XP593={X 1222,Y 549,Z -5,A 0,B -90,C 180,S 6,T 16,E1 0.0,E2 0.0,E3 0.0,E4 0.0,E5 0.0,E6 0.0}
DECL FDAT FP593={TOOL_NO 4,BASE_NO 0,IPO_FRAME #BASE,POINT2[] " "}
DECL LDAT LCPDAT593={VEL 1,ACC 50.000,APO_DIST 500.000,APO_FAC 50.0000,AXIS_VEL 50.000,AXIS_ACC 50.000,ORI_TYP #VAR,CIRC_TYP #BASE,JERK_FAC 50.0000,GEAR_JERK 100.000,EXAX_IGN 0}

DECL E6POS XP594={X 1272,Y 549,Z -5,A 0,B -90,C 180,S 6,T 16,E1 0.0,E2 0.0,E3 0.0,E4 0.0,E5 0.0,E6 0.0}
DECL FDAT FP594={TOOL_NO 4,BASE_NO 0,IPO_FRAME #BASE,POINT2[] " "}
DECL LDAT LCPDAT594={VEL 1,ACC 50.000,APO_DIST 500.000,APO_FAC 50.0000,AXIS_VEL 50.000,AXIS_ACC 50.000,ORI_TYP #VAR,CIRC_TYP #BASE,JERK_FAC 50.0000,GEAR_JERK 100.000,EXAX_IGN 0}

DECL E6POS XP595={X 1272,Y 549,Z 45,A 0,B -90,C 180,S 6,T 16,E1 0.0,E2 0.0,E3 0.0,E4 0.0,E5 0.0,E6 0.0}
DECL FDAT FP595={TOOL_NO 4,BASE_NO 0,IPO_FRAME #BASE,POINT2[] " "}
DECL LDAT LCPDAT595={VEL 1,ACC 50.000,APO_DIST 500.000,APO_FAC 50.0000,AXIS_VEL 50.000,AXIS_ACC 50.000,ORI_TYP #VAR,CIRC_TYP #BASE,JERK_FAC 50.0000,GEAR_JERK 100.000,EXAX_IGN 0}

DECL E6POS XP596={X 1222,Y 549,Z 45,A 0,B -90,C 180,S 6,T 16,E1 0.0,E2 0.0,E3 0.0,E4 0.0,E5 0.0,E6 0.0}
DECL FDAT FP596={TOOL_NO 4,BASE_NO 0,IPO_FRAME #BASE,POINT2[] " "}
DECL LDAT LCPDAT596={VEL 1,ACC 50.000,APO_DIST 500.000,APO_FAC 50.0000,AXIS_VEL 50.000,AXIS_ACC 50.000,ORI_TYP #VAR,CIRC_TYP #BASE,JERK_FAC 50.0000,GEAR_JERK 100.000,EXAX_IGN 0}

DECL E6POS XP597={X 1172,Y 549,Z 45,A 0,B -90,C 180,S 6,T 16,E1 0.0,E2 0.0,E3 0.0,E4 0.0,E5 0.0,E6 0.0}
DECL FDAT FP597={TOOL_NO 4,BASE_NO 0,IPO_FRAME #BASE,POINT2[] " "}
DECL LDAT LCPDAT597={VEL 1,ACC 50.000,APO_DIST 500.000,APO_FAC 50.0000,AXIS_VEL 50.000,AXIS_ACC 50.000,ORI_TYP #VAR,CIRC_TYP #BASE,JERK_FAC 50.0000,GEAR_JERK 100.000,EXAX_IGN 0}

DECL E6POS XP598={X 1122,Y 549,Z 45,A 0,B -90,C 180,S 6,T 16,E1 0.0,E2 0.0,E3 0.0,E4 0.0,E5 0.0,E6 0.0}
DECL FDAT FP598={TOOL_NO 4,BASE_NO 0,IPO_FRAME #BASE,POINT2[] " "}
DECL LDAT LCPDAT598={VEL 1,ACC 50.000,APO_DIST 500.000,APO_FAC 50.0000,AXIS_VEL 50.000,AXIS_ACC 50.000,ORI_TYP #VAR,CIRC_TYP #BASE,JERK_FAC 50.0000,GEAR_JERK 100.000,EXAX_IGN 0}

DECL E6POS XP599={X 1072,Y 549,Z 45,A 0,B -90,C 180,S 6,T 16,E1 0.0,E2 0.0,E3 0.0,E4 0.0,E5 0.0,E6 0.0}
DECL FDAT FP599={TOOL_NO 4,BASE_NO 0,IPO_FRAME #BASE,POINT2[] " "}
DECL LDAT LCPDAT599={VEL 1,ACC 50.000,APO_DIST 500.000,APO_FAC 50.0000,AXIS_VEL 50.000,AXIS_ACC 50.000,ORI_TYP #VAR,CIRC_TYP #BASE,JERK_FAC 50.0000,GEAR_JERK 100.000,EXAX_IGN 0}

DECL E6POS XP600={X 1022,Y 549,Z 45,A 0,B -90,C 180,S 6,T 16,E1 0.0,E2 0.0,E3 0.0,E4 0.0,E5 0.0,E6 0.0}
DECL FDAT FP600={TOOL_NO 4,BASE_NO 0,IPO_FRAME #BASE,POINT2[] " "}
DECL LDAT LCPDAT600={VEL 1,ACC 50.000,APO_DIST 500.000,APO_FAC 50.0000,AXIS_VEL 50.000,AXIS_ACC 50.000,ORI_TYP #VAR,CIRC_TYP #BASE,JERK_FAC 50.0000,GEAR_JERK 100.000,EXAX_IGN 0}

DECL E6POS XP601={X 972,Y 549,Z 45,A 0,B -90,C 180,S 6,T 16,E1 0.0,E2 0.0,E3 0.0,E4 0.0,E5 0.0,E6 0.0}
DECL FDAT FP601={TOOL_NO 4,BASE_NO 0,IPO_FRAME #BASE,POINT2[] " "}
DECL LDAT LCPDAT601={VEL 1,ACC 50.000,APO_DIST 500.000,APO_FAC 50.0000,AXIS_VEL 50.000,AXIS_ACC 50.000,ORI_TYP #VAR,CIRC_TYP #BASE,JERK_FAC 50.0000,GEAR_JERK 100.000,EXAX_IGN 0}

DECL E6POS XP602={X 922,Y 549,Z 45,A 0,B -90,C 180,S 6,T 16,E1 0.0,E2 0.0,E3 0.0,E4 0.0,E5 0.0,E6 0.0}
DECL FDAT FP602={TOOL_NO 4,BASE_NO 0,IPO_FRAME #BASE,POINT2[] " "}
DECL LDAT LCPDAT602={VEL 1,ACC 50.000,APO_DIST 500.000,APO_FAC 50.0000,AXIS_VEL 50.000,AXIS_ACC 50.000,ORI_TYP #VAR,CIRC_TYP #BASE,JERK_FAC 50.0000,GEAR_JERK 100.000,EXAX_IGN 0}

DECL E6POS XP603={X 872,Y 549,Z 45,A 0,B -90,C 180,S 6,T 16,E1 0.0,E2 0.0,E3 0.0,E4 0.0,E5 0.0,E6 0.0}
DECL FDAT FP603={TOOL_NO 4,BASE_NO 0,IPO_FRAME #BASE,POINT2[] " "}
DECL LDAT LCPDAT603={VEL 1,ACC 50.000,APO_DIST 500.000,APO_FAC 50.0000,AXIS_VEL 50.000,AXIS_ACC 50.000,ORI_TYP #VAR,CIRC_TYP #BASE,JERK_FAC 50.0000,GEAR_JERK 100.000,EXAX_IGN 0}

DECL E6POS XP604={X 822,Y 549,Z 45,A 0,B -90,C 180,S 6,T 16,E1 0.0,E2 0.0,E3 0.0,E4 0.0,E5 0.0,E6 0.0}
DECL FDAT FP604={TOOL_NO 4,BASE_NO 0,IPO_FRAME #BASE,POINT2[] " "}
DECL LDAT LCPDAT604={VEL 1,ACC 50.000,APO_DIST 500.000,APO_FAC 50.0000,AXIS_VEL 50.000,AXIS_ACC 50.000,ORI_TYP #VAR,CIRC_TYP #BASE,JERK_FAC 50.0000,GEAR_JERK 100.000,EXAX_IGN 0}

DECL E6POS XP605={X 772,Y 549,Z 45,A 0,B -90,C 180,S 6,T 16,E1 0.0,E2 0.0,E3 0.0,E4 0.0,E5 0.0,E6 0.0}
DECL FDAT FP605={TOOL_NO 4,BASE_NO 0,IPO_FRAME #BASE,POINT2[] " "}
DECL LDAT LCPDAT605={VEL 1,ACC 50.000,APO_DIST 500.000,APO_FAC 50.0000,AXIS_VEL 50.000,AXIS_ACC 50.000,ORI_TYP #VAR,CIRC_TYP #BASE,JERK_FAC 50.0000,GEAR_JERK 100.000,EXAX_IGN 0}

DECL E6POS XP606={X 722,Y 549,Z 45,A 0,B -90,C 180,S 6,T 16,E1 0.0,E2 0.0,E3 0.0,E4 0.0,E5 0.0,E6 0.0}
DECL FDAT FP606={TOOL_NO 4,BASE_NO 0,IPO_FRAME #BASE,POINT2[] " "}
DECL LDAT LCPDAT606={VEL 1,ACC 50.000,APO_DIST 500.000,APO_FAC 50.0000,AXIS_VEL 50.000,AXIS_ACC 50.000,ORI_TYP #VAR,CIRC_TYP #BASE,JERK_FAC 50.0000,GEAR_JERK 100.000,EXAX_IGN 0}

DECL E6POS XP607={X 672,Y 549,Z 45,A 0,B -90,C 180,S 6,T 16,E1 0.0,E2 0.0,E3 0.0,E4 0.0,E5 0.0,E6 0.0}
DECL FDAT FP607={TOOL_NO 4,BASE_NO 0,IPO_FRAME #BASE,POINT2[] " "}
DECL LDAT LCPDAT607={VEL 1,ACC 50.000,APO_DIST 500.000,APO_FAC 50.0000,AXIS_VEL 50.000,AXIS_ACC 50.000,ORI_TYP #VAR,CIRC_TYP #BASE,JERK_FAC 50.0000,GEAR_JERK 100.000,EXAX_IGN 0}

DECL E6POS XP608={X 672,Y 549,Z 95,A 0,B -90,C 180,S 6,T 16,E1 0.0,E2 0.0,E3 0.0,E4 0.0,E5 0.0,E6 0.0}
DECL FDAT FP608={TOOL_NO 4,BASE_NO 0,IPO_FRAME #BASE,POINT2[] " "}
DECL LDAT LCPDAT608={VEL 1,ACC 50.000,APO_DIST 500.000,APO_FAC 50.0000,AXIS_VEL 50.000,AXIS_ACC 50.000,ORI_TYP #VAR,CIRC_TYP #BASE,JERK_FAC 50.0000,GEAR_JERK 100.000,EXAX_IGN 0}

DECL E6POS XP609={X 722,Y 549,Z 95,A 0,B -90,C 180,S 6,T 16,E1 0.0,E2 0.0,E3 0.0,E4 0.0,E5 0.0,E6 0.0}
DECL FDAT FP609={TOOL_NO 4,BASE_NO 0,IPO_FRAME #BASE,POINT2[] " "}
DECL LDAT LCPDAT609={VEL 1,ACC 50.000,APO_DIST 500.000,APO_FAC 50.0000,AXIS_VEL 50.000,AXIS_ACC 50.000,ORI_TYP #VAR,CIRC_TYP #BASE,JERK_FAC 50.0000,GEAR_JERK 100.000,EXAX_IGN 0}

DECL E6POS XP610={X 772,Y 549,Z 95,A 0,B -90,C 180,S 6,T 16,E1 0.0,E2 0.0,E3 0.0,E4 0.0,E5 0.0,E6 0.0}
DECL FDAT FP610={TOOL_NO 4,BASE_NO 0,IPO_FRAME #BASE,POINT2[] " "}
DECL LDAT LCPDAT610={VEL 1,ACC 50.000,APO_DIST 500.000,APO_FAC 50.0000,AXIS_VEL 50.000,AXIS_ACC 50.000,ORI_TYP #VAR,CIRC_TYP #BASE,JERK_FAC 50.0000,GEAR_JERK 100.000,EXAX_IGN 0}

DECL E6POS XP611={X 822,Y 549,Z 95,A 0,B -90,C 180,S 6,T 16,E1 0.0,E2 0.0,E3 0.0,E4 0.0,E5 0.0,E6 0.0}
DECL FDAT FP611={TOOL_NO 4,BASE_NO 0,IPO_FRAME #BASE,POINT2[] " "}
DECL LDAT LCPDAT611={VEL 1,ACC 50.000,APO_DIST 500.000,APO_FAC 50.0000,AXIS_VEL 50.000,AXIS_ACC 50.000,ORI_TYP #VAR,CIRC_TYP #BASE,JERK_FAC 50.0000,GEAR_JERK 100.000,EXAX_IGN 0}

DECL E6POS XP612={X 872,Y 549,Z 95,A 0,B -90,C 180,S 6,T 16,E1 0.0,E2 0.0,E3 0.0,E4 0.0,E5 0.0,E6 0.0}
DECL FDAT FP612={TOOL_NO 4,BASE_NO 0,IPO_FRAME #BASE,POINT2[] " "}
DECL LDAT LCPDAT612={VEL 1,ACC 50.000,APO_DIST 500.000,APO_FAC 50.0000,AXIS_VEL 50.000,AXIS_ACC 50.000,ORI_TYP #VAR,CIRC_TYP #BASE,JERK_FAC 50.0000,GEAR_JERK 100.000,EXAX_IGN 0}

DECL E6POS XP613={X 922,Y 549,Z 95,A 0,B -90,C 180,S 6,T 16,E1 0.0,E2 0.0,E3 0.0,E4 0.0,E5 0.0,E6 0.0}
DECL FDAT FP613={TOOL_NO 4,BASE_NO 0,IPO_FRAME #BASE,POINT2[] " "}
DECL LDAT LCPDAT613={VEL 1,ACC 50.000,APO_DIST 500.000,APO_FAC 50.0000,AXIS_VEL 50.000,AXIS_ACC 50.000,ORI_TYP #VAR,CIRC_TYP #BASE,JERK_FAC 50.0000,GEAR_JERK 100.000,EXAX_IGN 0}

DECL E6POS XP614={X 972,Y 549,Z 95,A 0,B -90,C 180,S 6,T 16,E1 0.0,E2 0.0,E3 0.0,E4 0.0,E5 0.0,E6 0.0}
DECL FDAT FP614={TOOL_NO 4,BASE_NO 0,IPO_FRAME #BASE,POINT2[] " "}
DECL LDAT LCPDAT614={VEL 1,ACC 50.000,APO_DIST 500.000,APO_FAC 50.0000,AXIS_VEL 50.000,AXIS_ACC 50.000,ORI_TYP #VAR,CIRC_TYP #BASE,JERK_FAC 50.0000,GEAR_JERK 100.000,EXAX_IGN 0}

DECL E6POS XP615={X 1022,Y 549,Z 95,A 0,B -90,C 180,S 6,T 16,E1 0.0,E2 0.0,E3 0.0,E4 0.0,E5 0.0,E6 0.0}
DECL FDAT FP615={TOOL_NO 4,BASE_NO 0,IPO_FRAME #BASE,POINT2[] " "}
DECL LDAT LCPDAT615={VEL 1,ACC 50.000,APO_DIST 500.000,APO_FAC 50.0000,AXIS_VEL 50.000,AXIS_ACC 50.000,ORI_TYP #VAR,CIRC_TYP #BASE,JERK_FAC 50.0000,GEAR_JERK 100.000,EXAX_IGN 0}

DECL E6POS XP616={X 1072,Y 549,Z 95,A 0,B -90,C 180,S 6,T 16,E1 0.0,E2 0.0,E3 0.0,E4 0.0,E5 0.0,E6 0.0}
DECL FDAT FP616={TOOL_NO 4,BASE_NO 0,IPO_FRAME #BASE,POINT2[] " "}
DECL LDAT LCPDAT616={VEL 1,ACC 50.000,APO_DIST 500.000,APO_FAC 50.0000,AXIS_VEL 50.000,AXIS_ACC 50.000,ORI_TYP #VAR,CIRC_TYP #BASE,JERK_FAC 50.0000,GEAR_JERK 100.000,EXAX_IGN 0}

DECL E6POS XP617={X 1122,Y 549,Z 95,A 0,B -90,C 180,S 6,T 16,E1 0.0,E2 0.0,E3 0.0,E4 0.0,E5 0.0,E6 0.0}
DECL FDAT FP617={TOOL_NO 4,BASE_NO 0,IPO_FRAME #BASE,POINT2[] " "}
DECL LDAT LCPDAT617={VEL 1,ACC 50.000,APO_DIST 500.000,APO_FAC 50.0000,AXIS_VEL 50.000,AXIS_ACC 50.000,ORI_TYP #VAR,CIRC_TYP #BASE,JERK_FAC 50.0000,GEAR_JERK 100.000,EXAX_IGN 0}

DECL E6POS XP618={X 1172,Y 549,Z 95,A 0,B -90,C 180,S 6,T 16,E1 0.0,E2 0.0,E3 0.0,E4 0.0,E5 0.0,E6 0.0}
DECL FDAT FP618={TOOL_NO 4,BASE_NO 0,IPO_FRAME #BASE,POINT2[] " "}
DECL LDAT LCPDAT618={VEL 1,ACC 50.000,APO_DIST 500.000,APO_FAC 50.0000,AXIS_VEL 50.000,AXIS_ACC 50.000,ORI_TYP #VAR,CIRC_TYP #BASE,JERK_FAC 50.0000,GEAR_JERK 100.000,EXAX_IGN 0}

DECL E6POS XP619={X 1222,Y 549,Z 95,A 0,B -90,C 180,S 6,T 16,E1 0.0,E2 0.0,E3 0.0,E4 0.0,E5 0.0,E6 0.0}
DECL FDAT FP619={TOOL_NO 4,BASE_NO 0,IPO_FRAME #BASE,POINT2[] " "}
DECL LDAT LCPDAT619={VEL 1,ACC 50.000,APO_DIST 500.000,APO_FAC 50.0000,AXIS_VEL 50.000,AXIS_ACC 50.000,ORI_TYP #VAR,CIRC_TYP #BASE,JERK_FAC 50.0000,GEAR_JERK 100.000,EXAX_IGN 0}

DECL E6POS XP620={X 1272,Y 549,Z 95,A 0,B -90,C 180,S 6,T 16,E1 0.0,E2 0.0,E3 0.0,E4 0.0,E5 0.0,E6 0.0}
DECL FDAT FP620={TOOL_NO 4,BASE_NO 0,IPO_FRAME #BASE,POINT2[] " "}
DECL LDAT LCPDAT620={VEL 1,ACC 50.000,APO_DIST 500.000,APO_FAC 50.0000,AXIS_VEL 50.000,AXIS_ACC 50.000,ORI_TYP #VAR,CIRC_TYP #BASE,JERK_FAC 50.0000,GEAR_JERK 100.000,EXAX_IGN 0}

DECL E6POS XP621={X 1272,Y 549,Z 145,A 0,B -90,C 180,S 6,T 16,E1 0.0,E2 0.0,E3 0.0,E4 0.0,E5 0.0,E6 0.0}
DECL FDAT FP621={TOOL_NO 4,BASE_NO 0,IPO_FRAME #BASE,POINT2[] " "}
DECL LDAT LCPDAT621={VEL 1,ACC 50.000,APO_DIST 500.000,APO_FAC 50.0000,AXIS_VEL 50.000,AXIS_ACC 50.000,ORI_TYP #VAR,CIRC_TYP #BASE,JERK_FAC 50.0000,GEAR_JERK 100.000,EXAX_IGN 0}

DECL E6POS XP622={X 1222,Y 549,Z 145,A 0,B -90,C 180,S 6,T 16,E1 0.0,E2 0.0,E3 0.0,E4 0.0,E5 0.0,E6 0.0}
DECL FDAT FP622={TOOL_NO 4,BASE_NO 0,IPO_FRAME #BASE,POINT2[] " "}
DECL LDAT LCPDAT622={VEL 1,ACC 50.000,APO_DIST 500.000,APO_FAC 50.0000,AXIS_VEL 50.000,AXIS_ACC 50.000,ORI_TYP #VAR,CIRC_TYP #BASE,JERK_FAC 50.0000,GEAR_JERK 100.000,EXAX_IGN 0}

DECL E6POS XP623={X 1172,Y 549,Z 145,A 0,B -90,C 180,S 6,T 16,E1 0.0,E2 0.0,E3 0.0,E4 0.0,E5 0.0,E6 0.0}
DECL FDAT FP623={TOOL_NO 4,BASE_NO 0,IPO_FRAME #BASE,POINT2[] " "}
DECL LDAT LCPDAT623={VEL 1,ACC 50.000,APO_DIST 500.000,APO_FAC 50.0000,AXIS_VEL 50.000,AXIS_ACC 50.000,ORI_TYP #VAR,CIRC_TYP #BASE,JERK_FAC 50.0000,GEAR_JERK 100.000,EXAX_IGN 0}

DECL E6POS XP624={X 1122,Y 549,Z 145,A 0,B -90,C 180,S 6,T 16,E1 0.0,E2 0.0,E3 0.0,E4 0.0,E5 0.0,E6 0.0}
DECL FDAT FP624={TOOL_NO 4,BASE_NO 0,IPO_FRAME #BASE,POINT2[] " "}
DECL LDAT LCPDAT624={VEL 1,ACC 50.000,APO_DIST 500.000,APO_FAC 50.0000,AXIS_VEL 50.000,AXIS_ACC 50.000,ORI_TYP #VAR,CIRC_TYP #BASE,JERK_FAC 50.0000,GEAR_JERK 100.000,EXAX_IGN 0}

DECL E6POS XP625={X 1072,Y 549,Z 145,A 0,B -90,C 180,S 6,T 16,E1 0.0,E2 0.0,E3 0.0,E4 0.0,E5 0.0,E6 0.0}
DECL FDAT FP625={TOOL_NO 4,BASE_NO 0,IPO_FRAME #BASE,POINT2[] " "}
DECL LDAT LCPDAT625={VEL 1,ACC 50.000,APO_DIST 500.000,APO_FAC 50.0000,AXIS_VEL 50.000,AXIS_ACC 50.000,ORI_TYP #VAR,CIRC_TYP #BASE,JERK_FAC 50.0000,GEAR_JERK 100.000,EXAX_IGN 0}

DECL E6POS XP626={X 1022,Y 549,Z 145,A 0,B -90,C 180,S 6,T 16,E1 0.0,E2 0.0,E3 0.0,E4 0.0,E5 0.0,E6 0.0}
DECL FDAT FP626={TOOL_NO 4,BASE_NO 0,IPO_FRAME #BASE,POINT2[] " "}
DECL LDAT LCPDAT626={VEL 1,ACC 50.000,APO_DIST 500.000,APO_FAC 50.0000,AXIS_VEL 50.000,AXIS_ACC 50.000,ORI_TYP #VAR,CIRC_TYP #BASE,JERK_FAC 50.0000,GEAR_JERK 100.000,EXAX_IGN 0}

DECL E6POS XP627={X 972,Y 549,Z 145,A 0,B -90,C 180,S 6,T 16,E1 0.0,E2 0.0,E3 0.0,E4 0.0,E5 0.0,E6 0.0}
DECL FDAT FP627={TOOL_NO 4,BASE_NO 0,IPO_FRAME #BASE,POINT2[] " "}
DECL LDAT LCPDAT627={VEL 1,ACC 50.000,APO_DIST 500.000,APO_FAC 50.0000,AXIS_VEL 50.000,AXIS_ACC 50.000,ORI_TYP #VAR,CIRC_TYP #BASE,JERK_FAC 50.0000,GEAR_JERK 100.000,EXAX_IGN 0}

DECL E6POS XP628={X 922,Y 549,Z 145,A 0,B -90,C 180,S 6,T 16,E1 0.0,E2 0.0,E3 0.0,E4 0.0,E5 0.0,E6 0.0}
DECL FDAT FP628={TOOL_NO 4,BASE_NO 0,IPO_FRAME #BASE,POINT2[] " "}
DECL LDAT LCPDAT628={VEL 1,ACC 50.000,APO_DIST 500.000,APO_FAC 50.0000,AXIS_VEL 50.000,AXIS_ACC 50.000,ORI_TYP #VAR,CIRC_TYP #BASE,JERK_FAC 50.0000,GEAR_JERK 100.000,EXAX_IGN 0}

DECL E6POS XP629={X 872,Y 549,Z 145,A 0,B -90,C 180,S 6,T 16,E1 0.0,E2 0.0,E3 0.0,E4 0.0,E5 0.0,E6 0.0}
DECL FDAT FP629={TOOL_NO 4,BASE_NO 0,IPO_FRAME #BASE,POINT2[] " "}
DECL LDAT LCPDAT629={VEL 1,ACC 50.000,APO_DIST 500.000,APO_FAC 50.0000,AXIS_VEL 50.000,AXIS_ACC 50.000,ORI_TYP #VAR,CIRC_TYP #BASE,JERK_FAC 50.0000,GEAR_JERK 100.000,EXAX_IGN 0}

DECL E6POS XP630={X 822,Y 549,Z 145,A 0,B -90,C 180,S 6,T 16,E1 0.0,E2 0.0,E3 0.0,E4 0.0,E5 0.0,E6 0.0}
DECL FDAT FP630={TOOL_NO 4,BASE_NO 0,IPO_FRAME #BASE,POINT2[] " "}
DECL LDAT LCPDAT630={VEL 1,ACC 50.000,APO_DIST 500.000,APO_FAC 50.0000,AXIS_VEL 50.000,AXIS_ACC 50.000,ORI_TYP #VAR,CIRC_TYP #BASE,JERK_FAC 50.0000,GEAR_JERK 100.000,EXAX_IGN 0}

DECL E6POS XP631={X 772,Y 549,Z 145,A 0,B -90,C 180,S 6,T 16,E1 0.0,E2 0.0,E3 0.0,E4 0.0,E5 0.0,E6 0.0}
DECL FDAT FP631={TOOL_NO 4,BASE_NO 0,IPO_FRAME #BASE,POINT2[] " "}
DECL LDAT LCPDAT631={VEL 1,ACC 50.000,APO_DIST 500.000,APO_FAC 50.0000,AXIS_VEL 50.000,AXIS_ACC 50.000,ORI_TYP #VAR,CIRC_TYP #BASE,JERK_FAC 50.0000,GEAR_JERK 100.000,EXAX_IGN 0}

DECL E6POS XP632={X 722,Y 549,Z 145,A 0,B -90,C 180,S 6,T 16,E1 0.0,E2 0.0,E3 0.0,E4 0.0,E5 0.0,E6 0.0}
DECL FDAT FP632={TOOL_NO 4,BASE_NO 0,IPO_FRAME #BASE,POINT2[] " "}
DECL LDAT LCPDAT632={VEL 1,ACC 50.000,APO_DIST 500.000,APO_FAC 50.0000,AXIS_VEL 50.000,AXIS_ACC 50.000,ORI_TYP #VAR,CIRC_TYP #BASE,JERK_FAC 50.0000,GEAR_JERK 100.000,EXAX_IGN 0}

DECL E6POS XP633={X 672,Y 549,Z 145,A 0,B -90,C 180,S 6,T 16,E1 0.0,E2 0.0,E3 0.0,E4 0.0,E5 0.0,E6 0.0}
DECL FDAT FP633={TOOL_NO 4,BASE_NO 0,IPO_FRAME #BASE,POINT2[] " "}
DECL LDAT LCPDAT633={VEL 1,ACC 50.000,APO_DIST 500.000,APO_FAC 50.0000,AXIS_VEL 50.000,AXIS_ACC 50.000,ORI_TYP #VAR,CIRC_TYP #BASE,JERK_FAC 50.0000,GEAR_JERK 100.000,EXAX_IGN 0}

DECL E6POS XP634={X 672,Y 549,Z 195,A 0,B -90,C 180,S 6,T 16,E1 0.0,E2 0.0,E3 0.0,E4 0.0,E5 0.0,E6 0.0}
DECL FDAT FP634={TOOL_NO 4,BASE_NO 0,IPO_FRAME #BASE,POINT2[] " "}
DECL LDAT LCPDAT634={VEL 1,ACC 50.000,APO_DIST 500.000,APO_FAC 50.0000,AXIS_VEL 50.000,AXIS_ACC 50.000,ORI_TYP #VAR,CIRC_TYP #BASE,JERK_FAC 50.0000,GEAR_JERK 100.000,EXAX_IGN 0}

DECL E6POS XP635={X 722,Y 549,Z 195,A 0,B -90,C 180,S 6,T 16,E1 0.0,E2 0.0,E3 0.0,E4 0.0,E5 0.0,E6 0.0}
DECL FDAT FP635={TOOL_NO 4,BASE_NO 0,IPO_FRAME #BASE,POINT2[] " "}
DECL LDAT LCPDAT635={VEL 1,ACC 50.000,APO_DIST 500.000,APO_FAC 50.0000,AXIS_VEL 50.000,AXIS_ACC 50.000,ORI_TYP #VAR,CIRC_TYP #BASE,JERK_FAC 50.0000,GEAR_JERK 100.000,EXAX_IGN 0}

DECL E6POS XP636={X 772,Y 549,Z 195,A 0,B -90,C 180,S 6,T 16,E1 0.0,E2 0.0,E3 0.0,E4 0.0,E5 0.0,E6 0.0}
DECL FDAT FP636={TOOL_NO 4,BASE_NO 0,IPO_FRAME #BASE,POINT2[] " "}
DECL LDAT LCPDAT636={VEL 1,ACC 50.000,APO_DIST 500.000,APO_FAC 50.0000,AXIS_VEL 50.000,AXIS_ACC 50.000,ORI_TYP #VAR,CIRC_TYP #BASE,JERK_FAC 50.0000,GEAR_JERK 100.000,EXAX_IGN 0}

DECL E6POS XP637={X 822,Y 549,Z 195,A 0,B -90,C 180,S 6,T 16,E1 0.0,E2 0.0,E3 0.0,E4 0.0,E5 0.0,E6 0.0}
DECL FDAT FP637={TOOL_NO 4,BASE_NO 0,IPO_FRAME #BASE,POINT2[] " "}
DECL LDAT LCPDAT637={VEL 1,ACC 50.000,APO_DIST 500.000,APO_FAC 50.0000,AXIS_VEL 50.000,AXIS_ACC 50.000,ORI_TYP #VAR,CIRC_TYP #BASE,JERK_FAC 50.0000,GEAR_JERK 100.000,EXAX_IGN 0}

DECL E6POS XP638={X 872,Y 549,Z 195,A 0,B -90,C 180,S 6,T 16,E1 0.0,E2 0.0,E3 0.0,E4 0.0,E5 0.0,E6 0.0}
DECL FDAT FP638={TOOL_NO 4,BASE_NO 0,IPO_FRAME #BASE,POINT2[] " "}
DECL LDAT LCPDAT638={VEL 1,ACC 50.000,APO_DIST 500.000,APO_FAC 50.0000,AXIS_VEL 50.000,AXIS_ACC 50.000,ORI_TYP #VAR,CIRC_TYP #BASE,JERK_FAC 50.0000,GEAR_JERK 100.000,EXAX_IGN 0}

DECL E6POS XP639={X 922,Y 549,Z 195,A 0,B -90,C 180,S 6,T 16,E1 0.0,E2 0.0,E3 0.0,E4 0.0,E5 0.0,E6 0.0}
DECL FDAT FP639={TOOL_NO 4,BASE_NO 0,IPO_FRAME #BASE,POINT2[] " "}
DECL LDAT LCPDAT639={VEL 1,ACC 50.000,APO_DIST 500.000,APO_FAC 50.0000,AXIS_VEL 50.000,AXIS_ACC 50.000,ORI_TYP #VAR,CIRC_TYP #BASE,JERK_FAC 50.0000,GEAR_JERK 100.000,EXAX_IGN 0}

DECL E6POS XP640={X 972,Y 549,Z 195,A 0,B -90,C 180,S 6,T 16,E1 0.0,E2 0.0,E3 0.0,E4 0.0,E5 0.0,E6 0.0}
DECL FDAT FP640={TOOL_NO 4,BASE_NO 0,IPO_FRAME #BASE,POINT2[] " "}
DECL LDAT LCPDAT640={VEL 1,ACC 50.000,APO_DIST 500.000,APO_FAC 50.0000,AXIS_VEL 50.000,AXIS_ACC 50.000,ORI_TYP #VAR,CIRC_TYP #BASE,JERK_FAC 50.0000,GEAR_JERK 100.000,EXAX_IGN 0}

DECL E6POS XP641={X 1022,Y 549,Z 195,A 0,B -90,C 180,S 6,T 16,E1 0.0,E2 0.0,E3 0.0,E4 0.0,E5 0.0,E6 0.0}
DECL FDAT FP641={TOOL_NO 4,BASE_NO 0,IPO_FRAME #BASE,POINT2[] " "}
DECL LDAT LCPDAT641={VEL 1,ACC 50.000,APO_DIST 500.000,APO_FAC 50.0000,AXIS_VEL 50.000,AXIS_ACC 50.000,ORI_TYP #VAR,CIRC_TYP #BASE,JERK_FAC 50.0000,GEAR_JERK 100.000,EXAX_IGN 0}

DECL E6POS XP642={X 1072,Y 549,Z 195,A 0,B -90,C 180,S 6,T 16,E1 0.0,E2 0.0,E3 0.0,E4 0.0,E5 0.0,E6 0.0}
DECL FDAT FP642={TOOL_NO 4,BASE_NO 0,IPO_FRAME #BASE,POINT2[] " "}
DECL LDAT LCPDAT642={VEL 1,ACC 50.000,APO_DIST 500.000,APO_FAC 50.0000,AXIS_VEL 50.000,AXIS_ACC 50.000,ORI_TYP #VAR,CIRC_TYP #BASE,JERK_FAC 50.0000,GEAR_JERK 100.000,EXAX_IGN 0}

DECL E6POS XP643={X 1122,Y 549,Z 195,A 0,B -90,C 180,S 6,T 16,E1 0.0,E2 0.0,E3 0.0,E4 0.0,E5 0.0,E6 0.0}
DECL FDAT FP643={TOOL_NO 4,BASE_NO 0,IPO_FRAME #BASE,POINT2[] " "}
DECL LDAT LCPDAT643={VEL 1,ACC 50.000,APO_DIST 500.000,APO_FAC 50.0000,AXIS_VEL 50.000,AXIS_ACC 50.000,ORI_TYP #VAR,CIRC_TYP #BASE,JERK_FAC 50.0000,GEAR_JERK 100.000,EXAX_IGN 0}

DECL E6POS XP644={X 1172,Y 549,Z 195,A 0,B -90,C 180,S 6,T 16,E1 0.0,E2 0.0,E3 0.0,E4 0.0,E5 0.0,E6 0.0}
DECL FDAT FP644={TOOL_NO 4,BASE_NO 0,IPO_FRAME #BASE,POINT2[] " "}
DECL LDAT LCPDAT644={VEL 1,ACC 50.000,APO_DIST 500.000,APO_FAC 50.0000,AXIS_VEL 50.000,AXIS_ACC 50.000,ORI_TYP #VAR,CIRC_TYP #BASE,JERK_FAC 50.0000,GEAR_JERK 100.000,EXAX_IGN 0}

DECL E6POS XP645={X 1222,Y 549,Z 195,A 0,B -90,C 180,S 6,T 16,E1 0.0,E2 0.0,E3 0.0,E4 0.0,E5 0.0,E6 0.0}
DECL FDAT FP645={TOOL_NO 4,BASE_NO 0,IPO_FRAME #BASE,POINT2[] " "}
DECL LDAT LCPDAT645={VEL 1,ACC 50.000,APO_DIST 500.000,APO_FAC 50.0000,AXIS_VEL 50.000,AXIS_ACC 50.000,ORI_TYP #VAR,CIRC_TYP #BASE,JERK_FAC 50.0000,GEAR_JERK 100.000,EXAX_IGN 0}

DECL E6POS XP646={X 1272,Y 549,Z 195,A 0,B -90,C 180,S 6,T 16,E1 0.0,E2 0.0,E3 0.0,E4 0.0,E5 0.0,E6 0.0}
DECL FDAT FP646={TOOL_NO 4,BASE_NO 0,IPO_FRAME #BASE,POINT2[] " "}
DECL LDAT LCPDAT646={VEL 1,ACC 50.000,APO_DIST 500.000,APO_FAC 50.0000,AXIS_VEL 50.000,AXIS_ACC 50.000,ORI_TYP #VAR,CIRC_TYP #BASE,JERK_FAC 50.0000,GEAR_JERK 100.000,EXAX_IGN 0}

DECL E6POS XP647={X 1272,Y 549,Z 245,A 0,B -90,C 180,S 6,T 16,E1 0.0,E2 0.0,E3 0.0,E4 0.0,E5 0.0,E6 0.0}
DECL FDAT FP647={TOOL_NO 4,BASE_NO 0,IPO_FRAME #BASE,POINT2[] " "}
DECL LDAT LCPDAT647={VEL 1,ACC 50.000,APO_DIST 500.000,APO_FAC 50.0000,AXIS_VEL 50.000,AXIS_ACC 50.000,ORI_TYP #VAR,CIRC_TYP #BASE,JERK_FAC 50.0000,GEAR_JERK 100.000,EXAX_IGN 0}

DECL E6POS XP648={X 1222,Y 549,Z 245,A 0,B -90,C 180,S 6,T 16,E1 0.0,E2 0.0,E3 0.0,E4 0.0,E5 0.0,E6 0.0}
DECL FDAT FP648={TOOL_NO 4,BASE_NO 0,IPO_FRAME #BASE,POINT2[] " "}
DECL LDAT LCPDAT648={VEL 1,ACC 50.000,APO_DIST 500.000,APO_FAC 50.0000,AXIS_VEL 50.000,AXIS_ACC 50.000,ORI_TYP #VAR,CIRC_TYP #BASE,JERK_FAC 50.0000,GEAR_JERK 100.000,EXAX_IGN 0}

DECL E6POS XP649={X 1172,Y 549,Z 245,A 0,B -90,C 180,S 6,T 16,E1 0.0,E2 0.0,E3 0.0,E4 0.0,E5 0.0,E6 0.0}
DECL FDAT FP649={TOOL_NO 4,BASE_NO 0,IPO_FRAME #BASE,POINT2[] " "}
DECL LDAT LCPDAT649={VEL 1,ACC 50.000,APO_DIST 500.000,APO_FAC 50.0000,AXIS_VEL 50.000,AXIS_ACC 50.000,ORI_TYP #VAR,CIRC_TYP #BASE,JERK_FAC 50.0000,GEAR_JERK 100.000,EXAX_IGN 0}

DECL E6POS XP650={X 1122,Y 549,Z 245,A 0,B -90,C 180,S 6,T 16,E1 0.0,E2 0.0,E3 0.0,E4 0.0,E5 0.0,E6 0.0}
DECL FDAT FP650={TOOL_NO 4,BASE_NO 0,IPO_FRAME #BASE,POINT2[] " "}
DECL LDAT LCPDAT650={VEL 1,ACC 50.000,APO_DIST 500.000,APO_FAC 50.0000,AXIS_VEL 50.000,AXIS_ACC 50.000,ORI_TYP #VAR,CIRC_TYP #BASE,JERK_FAC 50.0000,GEAR_JERK 100.000,EXAX_IGN 0}

DECL E6POS XP651={X 1072,Y 549,Z 245,A 0,B -90,C 180,S 6,T 16,E1 0.0,E2 0.0,E3 0.0,E4 0.0,E5 0.0,E6 0.0}
DECL FDAT FP651={TOOL_NO 4,BASE_NO 0,IPO_FRAME #BASE,POINT2[] " "}
DECL LDAT LCPDAT651={VEL 1,ACC 50.000,APO_DIST 500.000,APO_FAC 50.0000,AXIS_VEL 50.000,AXIS_ACC 50.000,ORI_TYP #VAR,CIRC_TYP #BASE,JERK_FAC 50.0000,GEAR_JERK 100.000,EXAX_IGN 0}

DECL E6POS XP652={X 1022,Y 549,Z 245,A 0,B -90,C 180,S 6,T 16,E1 0.0,E2 0.0,E3 0.0,E4 0.0,E5 0.0,E6 0.0}
DECL FDAT FP652={TOOL_NO 4,BASE_NO 0,IPO_FRAME #BASE,POINT2[] " "}
DECL LDAT LCPDAT652={VEL 1,ACC 50.000,APO_DIST 500.000,APO_FAC 50.0000,AXIS_VEL 50.000,AXIS_ACC 50.000,ORI_TYP #VAR,CIRC_TYP #BASE,JERK_FAC 50.0000,GEAR_JERK 100.000,EXAX_IGN 0}

DECL E6POS XP653={X 972,Y 549,Z 245,A 0,B -90,C 180,S 6,T 16,E1 0.0,E2 0.0,E3 0.0,E4 0.0,E5 0.0,E6 0.0}
DECL FDAT FP653={TOOL_NO 4,BASE_NO 0,IPO_FRAME #BASE,POINT2[] " "}
DECL LDAT LCPDAT653={VEL 1,ACC 50.000,APO_DIST 500.000,APO_FAC 50.0000,AXIS_VEL 50.000,AXIS_ACC 50.000,ORI_TYP #VAR,CIRC_TYP #BASE,JERK_FAC 50.0000,GEAR_JERK 100.000,EXAX_IGN 0}

DECL E6POS XP654={X 922,Y 549,Z 245,A 0,B -90,C 180,S 6,T 16,E1 0.0,E2 0.0,E3 0.0,E4 0.0,E5 0.0,E6 0.0}
DECL FDAT FP654={TOOL_NO 4,BASE_NO 0,IPO_FRAME #BASE,POINT2[] " "}
DECL LDAT LCPDAT654={VEL 1,ACC 50.000,APO_DIST 500.000,APO_FAC 50.0000,AXIS_VEL 50.000,AXIS_ACC 50.000,ORI_TYP #VAR,CIRC_TYP #BASE,JERK_FAC 50.0000,GEAR_JERK 100.000,EXAX_IGN 0}

DECL E6POS XP655={X 872,Y 549,Z 245,A 0,B -90,C 180,S 6,T 16,E1 0.0,E2 0.0,E3 0.0,E4 0.0,E5 0.0,E6 0.0}
DECL FDAT FP655={TOOL_NO 4,BASE_NO 0,IPO_FRAME #BASE,POINT2[] " "}
DECL LDAT LCPDAT655={VEL 1,ACC 50.000,APO_DIST 500.000,APO_FAC 50.0000,AXIS_VEL 50.000,AXIS_ACC 50.000,ORI_TYP #VAR,CIRC_TYP #BASE,JERK_FAC 50.0000,GEAR_JERK 100.000,EXAX_IGN 0}

DECL E6POS XP656={X 822,Y 549,Z 245,A 0,B -90,C 180,S 6,T 16,E1 0.0,E2 0.0,E3 0.0,E4 0.0,E5 0.0,E6 0.0}
DECL FDAT FP656={TOOL_NO 4,BASE_NO 0,IPO_FRAME #BASE,POINT2[] " "}
DECL LDAT LCPDAT656={VEL 1,ACC 50.000,APO_DIST 500.000,APO_FAC 50.0000,AXIS_VEL 50.000,AXIS_ACC 50.000,ORI_TYP #VAR,CIRC_TYP #BASE,JERK_FAC 50.0000,GEAR_JERK 100.000,EXAX_IGN 0}

DECL E6POS XP657={X 772,Y 549,Z 245,A 0,B -90,C 180,S 6,T 16,E1 0.0,E2 0.0,E3 0.0,E4 0.0,E5 0.0,E6 0.0}
DECL FDAT FP657={TOOL_NO 4,BASE_NO 0,IPO_FRAME #BASE,POINT2[] " "}
DECL LDAT LCPDAT657={VEL 1,ACC 50.000,APO_DIST 500.000,APO_FAC 50.0000,AXIS_VEL 50.000,AXIS_ACC 50.000,ORI_TYP #VAR,CIRC_TYP #BASE,JERK_FAC 50.0000,GEAR_JERK 100.000,EXAX_IGN 0}

DECL E6POS XP658={X 722,Y 549,Z 245,A 0,B -90,C 180,S 6,T 16,E1 0.0,E2 0.0,E3 0.0,E4 0.0,E5 0.0,E6 0.0}
DECL FDAT FP658={TOOL_NO 4,BASE_NO 0,IPO_FRAME #BASE,POINT2[] " "}
DECL LDAT LCPDAT658={VEL 1,ACC 50.000,APO_DIST 500.000,APO_FAC 50.0000,AXIS_VEL 50.000,AXIS_ACC 50.000,ORI_TYP #VAR,CIRC_TYP #BASE,JERK_FAC 50.0000,GEAR_JERK 100.000,EXAX_IGN 0}

DECL E6POS XP659={X 672,Y 549,Z 245,A 0,B -90,C 180,S 6,T 16,E1 0.0,E2 0.0,E3 0.0,E4 0.0,E5 0.0,E6 0.0}
DECL FDAT FP659={TOOL_NO 4,BASE_NO 0,IPO_FRAME #BASE,POINT2[] " "}
DECL LDAT LCPDAT659={VEL 1,ACC 50.000,APO_DIST 500.000,APO_FAC 50.0000,AXIS_VEL 50.000,AXIS_ACC 50.000,ORI_TYP #VAR,CIRC_TYP #BASE,JERK_FAC 50.0000,GEAR_JERK 100.000,EXAX_IGN 0}

ENDDAT
